FUNCTION_BLOCK FB_DigitalOutput
VAR_INPUT
END_VAR
VAR_OUTPUT
END_VAR
VAR	
	// https://infosys.beckhoff.com/content/1033/tc3_plc_intro/11948825611.html?id=1756449079294237528
	Output AT %Q* : BOOL;
	_Output: BOOL;
	_FirstScan: BOOL;
END_VAR

IF _FirstScan THEN
	//
END_IF

// do some things?
Output :=_Output;

// do not put anything below this
_FirstScan := FALSE;

METHOD PUBLIC Off : BOOL
VAR_INPUT
END_VAR
_Output := FALSE;
END_METHOD

METHOD PUBLIC On : BOOL
VAR_INPUT
END_VAR
_Output := TRUE;
END_METHOD

{attribute 'monitoring' := 'variable'}
PROPERTY PUBLIC P_StateOff : BOOL
GET
P_StateOff := NOT _Output;
END_GET
END_PROPERTY

{attribute 'monitoring' := 'variable'}
PROPERTY PUBLIC P_StateOn : BOOL
GET
P_StateOn := _Output;
END_GET
END_PROPERTY

METHOD PUBLIC Toggle : BOOL
VAR_INPUT
END_VAR
_Output := NOT _Output;
END_METHOD

END_FUNCTION_BLOCK

(* stored: Version 1.1.0.1
   POU FB_DigitalOutput: Id {9ccb68c3-5dd7-4441-a68d-8f407a5bbf39}, SpecialFunc None
   Folder public: Id {0da57af1-9d70-4000-8a8d-dad5dfab92ff}
   Method Off: Id {f8b6fdb2-6544-4607-9a19-3594027652d2}
   Method On: Id {8d32d062-36c2-487a-8ff3-0192a0a033a4}
   Property P_StateOff: Id {e6661ae8-a7e9-466d-aa33-4575a19f892b}
   Get Get: Id {c5dfac2e-9fcf-40c5-98c6-a526c0fb2c0d}
   Property P_StateOn: Id {15ab277e-c978-4e7b-9e52-7a854e0469dd}
   Get Get: Id {3e9280db-f833-416e-8f4f-78f55b065785}
   Method Toggle: Id {acfd7b5d-3f2d-4ece-8bee-8a0616bd626e} *)
